  LIN {X -4860.893,Y -2029.899,Z -82.531,A 90.03341,B 0.00000,C 180.00000} ; retreat
  ; Step 3350, bar 1635
  LIN {X -4985.893,Y -2029.899,Z 855.478,A 90.03341,B 0.00000,C 180.00000} ; outside
  LIN {X -4985.893,Y -2029.899,Z -132.531,A 90.03341,B 0.00000,C 180.00000} ; preinsert
  LIN {X -4985.893,Y -2029.899,Z -382.531,A 90.03341,B 0.00000,C 180.00000} ; insert
  LIN {X -4985.893,Y -2029.899,Z -382.531,A 90.03341,B 0.00000,C 180.00000} ; release
  LIN {X -4985.893,Y -2029.899,Z -82.531,A 90.03341,B 0.00000,C 180.00000} ; retreat
  ; Step 3351, bar 1637
  LIN {X -5110.893,Y -2029.899,Z 855.478,A 90.03341,B 0.00000,C 180.00000} ; outside
  LIN {X -5110.893,Y -2029.899,Z -132.531,A 90.03341,B 0.00000,C 180.00000} ; preinsert
  LIN {X -5110.893,Y -2029.899,Z -382.531,A 90.03341,B 0.00000,C 180.00000} ; insert
  LIN {X -5110.893,Y -2029.899,Z -382.531,A 90.03341,B 0.00000,C 180.00000} ; release
  LIN {X -5110.893,Y -2029.899,Z -82.531,A 90.03341,B 0.00000,C 180.00000} ; retreat
  ; Step 3352, bar 1639
  LIN {X -5235.893,Y -2029.899,Z 855.478,A 90.03341,B 0.00000,C 180.00000} ; outside
  LIN {X -5235.893,Y -2029.899,Z -132.531,A 90.03341,B 0.00000,C 180.00000} ; preinsert
  LIN {X -5235.893,Y -2029.899,Z -382.531,A 90.03341,B 0.00000,C 180.00000} ; insert
  LIN {X -5235.893,Y -2029.899,Z -382.531,A 90.03341,B 0.00000,C 180.00000} ; release
  LIN {X -5235.893,Y -2029.899,Z -82.531,A 90.03341,B 0.00000,C 180.00000} ; retreat
  ; Step 3353, bar 1641
  LIN {X -5360.893,Y -2029.899,Z 855.478,A 90.03341,B 0.00000,C 180.00000} ; outside
  LIN {X -5360.893,Y -2029.899,Z -132.531,A 90.03341,B 0.00000,C 180.00000} ; preinsert
  LIN {X -5360.893,Y -2029.899,Z -382.531,A 90.03341,B 0.00000,C 180.00000} ; insert
  LIN {X -5360.893,Y -2029.899,Z -382.531,A 90.03341,B 0.00000,C 180.00000} ; release
  LIN {X -5360.893,Y -2029.899,Z -82.531,A 90.03341,B 0.00000,C 180.00000} ; retreat
  ; Step 3354, bar 1643
  LIN {X -5485.893,Y -2029.899,Z 855.478,A 90.03341,B 0.00000,C 180.00000} ; outside
  LIN {X -5485.893,Y -2029.899,Z -132.531,A 90.03341,B 0.00000,C 180.00000} ; preinsert
  LIN {X -5485.893,Y -2029.899,Z -382.531,A 90.03341,B 0.00000,C 180.00000} ; insert
  LIN {X -5485.893,Y -2029.899,Z -382.531,A 90.03341,B 0.00000,C 180.00000} ; release
  LIN {X -5485.893,Y -2029.899,Z -82.531,A 90.03341,B 0.00000,C 180.00000} ; retreat
  ; Step 3355, bar 1645
  LIN {X -5610.893,Y -2029.899,Z 855.478,A 90.03341,B 0.00000,C 180.00000} ; outside
  LIN {X -5610.893,Y -2029.899,Z -132.531,A 90.03341,B 0.00000,C 180.00000} ; preinsert
  LIN {X -5610.893,Y -2029.899,Z -382.531,A 90.03341,B 0.00000,C 180.00000} ; insert
  LIN {X -5610.893,Y -2029.899,Z -382.531,A 90.03341,B 0.00000,C 180.00000} ; release
  LIN {X -5610.893,Y -2029.899,Z -82.531,A 90.03341,B 0.00000,C 180.00000} ; retreat
  ; Step 3356, bar 1647
  LIN {X -5735.893,Y -2029.899,Z 855.478,A 90.03341,B 0.00000,C 180.00000} ; outside
  LIN {X -5735.893,Y -2029.899,Z -132.531,A 90.03341,B 0.00000,C 180.00000} ; preinsert
  LIN {X -5735.893,Y -2029.899,Z -382.531,A 90.03341,B 0.00000,C 180.00000} ; insert
  LIN {X -5735.893,Y -2029.899,Z -382.531,A 90.03341,B 0.00000,C 180.00000} ; release
  LIN {X -5735.893,Y -2029.899,Z -82.531,A 90.03341,B 0.00000,C 180.00000} ; retreat
  ; Step 3357, bar 1649
  LIN {X -5860.893,Y -2029.899,Z 855.478,A 90.03341,B 0.00000,C 180.00000} ; outside
  LIN {X -5860.893,Y -2029.899,Z -132.531,A 90.03341,B 0.00000,C 180.00000} ; preinsert
  LIN {X -5860.893,Y -2029.899,Z -382.531,A 90.03341,B 0.00000,C 180.00000} ; insert
  LIN {X -5860.893,Y -2029.899,Z -382.531,A 90.03341,B 0.00000,C 180.00000} ; release
  LIN {X -5860.893,Y -2029.899,Z -82.531,A 90.03341,B 0.00000,C 180.00000} ; retreat
  ; Step 3358, bar 1651
  LIN {X -6110.893,Y -2029.899,Z 855.478,A 90.03341,B 0.00000,C 180.00000} ; outside
  LIN {X -6110.893,Y -2029.899,Z -132.531,A 90.03341,B 0.00000,C 180.00000} ; preinsert
  LIN {X -6110.893,Y -2029.899,Z -382.531,A 90.03341,B 0.00000,C 180.00000} ; insert
  LIN {X -6110.893,Y -2029.899,Z -382.531,A 90.03341,B 0.00000,C 180.00000} ; release
  LIN {X -6110.893,Y -2029.899,Z -82.531,A 90.03341,B 0.00000,C 180.00000} ; retreat
  ; Step 3359, bar 1653
  LIN {X -6235.893,Y -2029.899,Z 855.478,A 90.03341,B 0.00000,C 180.00000} ; outside
  LIN {X -6235.893,Y -2029.899,Z -132.531,A 90.03341,B 0.00000,C 180.00000} ; preinsert
  LIN {X -6235.893,Y -2029.899,Z -382.531,A 90.03341,B 0.00000,C 180.00000} ; insert
  LIN {X -6235.893,Y -2029.899,Z -382.531,A 90.03341,B 0.00000,C 180.00000} ; release
  LIN {X -6235.893,Y -2029.899,Z -82.531,A 90.03341,B 0.00000,C 180.00000} ; retreat
  ; Step 3360, bar 1655
  LIN {X -6360.893,Y -2029.899,Z 855.478,A 90.03341,B 0.00000,C 180.00000} ; outside
  LIN {X -6360.893,Y -2029.899,Z -132.531,A 90.03341,B 0.00000,C 180.00000} ; preinsert
  LIN {X -6360.893,Y -2029.899,Z -382.531,A 90.03341,B 0.00000,C 180.00000} ; insert
  LIN {X -6360.893,Y -2029.899,Z -382.531,A 90.03341,B 0.00000,C 180.00000} ; release
  LIN {X -6360.893,Y -2029.899,Z -82.531,A 90.03341,B 0.00000,C 180.00000} ; retreat
  ; Step 3361, bar 1657
  LIN {X -6485.893,Y -2029.899,Z 855.478,A 90.03341,B 0.00000,C 180.00000} ; outside
  LIN {X -6485.893,Y -2029.899,Z -132.531,A 90.03341,B 0.00000,C 180.00000} ; preinsert
  LIN {X -6485.893,Y -2029.899,Z -382.531,A 90.03341,B 0.00000,C 180.00000} ; insert
  LIN {X -6485.893,Y -2029.899,Z -382.531,A 90.03341,B 0.00000,C 180.00000} ; release
  LIN {X -6485.893,Y -2029.899,Z -82.531,A 90.03341,B 0.00000,C 180.00000} ; retreat
  ; Step 3362, bar 1659
  LIN {X -6610.893,Y -2029.899,Z 855.478,A 90.03341,B 0.00000,C 180.00000} ; outside
  LIN {X -6610.893,Y -2029.899,Z -132.531,A 90.03341,B 0.00000,C 180.00000} ; preinsert
  LIN {X -6610.893,Y -2029.899,Z -382.531,A 90.03341,B 0.00000,C 180.00000} ; insert
  LIN {X -6610.893,Y -2029.899,Z -382.531,A 90.03341,B 0.00000,C 180.00000} ; release
  LIN {X -6610.893,Y -2029.899,Z -82.531,A 90.03341,B 0.00000,C 180.00000} ; retreat
  ; Step 3363, bar 1661
  LIN {X -6735.893,Y -2029.899,Z 855.478,A 90.03341,B 0.00000,C 180.00000} ; outside
  LIN {X -6735.893,Y -2029.899,Z -132.531,A 90.03341,B 0.00000,C 180.00000} ; preinsert
  LIN {X -6735.893,Y -2029.899,Z -382.531,A 90.03341,B 0.00000,C 180.00000} ; insert
  LIN {X -6735.893,Y -2029.899,Z -382.531,A 90.03341,B 0.00000,C 180.00000} ; release
  LIN {X -6735.893,Y -2029.899,Z -82.531,A 90.03341,B 0.00000,C 180.00000} ; retreat
  ; Step 3364, bar 1663
  LIN {X -6860.893,Y -2029.899,Z 855.478,A 90.03341,B 0.00000,C 180.00000} ; outside
  LIN {X -6860.893,Y -2029.899,Z -132.531,A 90.03341,B 0.00000,C 180.00000} ; preinsert
  LIN {X -6860.893,Y -2029.899,Z -382.531,A 90.03341,B 0.00000,C 180.00000} ; insert
  LIN {X -6860.893,Y -2029.899,Z -382.531,A 90.03341,B 0.00000,C 180.00000} ; release
  LIN {X -6860.893,Y -2029.899,Z -82.531,A 90.03341,B 0.00000,C 180.00000} ; retreat
  ; Step 3365, bar 1665
  LIN {X -6985.893,Y -2029.899,Z 855.478,A 90.03341,B 0.00000,C 180.00000} ; outside
  LIN {X -6985.893,Y -2029.899,Z -132.531,A 90.03341,B 0.00000,C 180.00000} ; preinsert
  LIN {X -6985.893,Y -2029.899,Z -382.531,A 90.03341,B 0.00000,C 180.00000} ; insert
  LIN {X -6985.893,Y -2029.899,Z -382.531,A 90.03341,B 0.00000,C 180.00000} ; release
  LIN {X -6985.893,Y -2029.899,Z -82.531,A 90.03341,B 0.00000,C 180.00000} ; retreat
  ; Step 3366, bar 1667
  LIN {X -7110.893,Y -2029.899,Z 855.478,A 90.03341,B 0.00000,C 180.00000} ; outside
  LIN {X -7110.893,Y -2029.899,Z -132.531,A 90.03341,B 0.00000,C 180.00000} ; preinsert
  LIN {X -7110.893,Y -2029.899,Z -382.531,A 90.03341,B 0.00000,C 180.00000} ; insert
  LIN {X -7110.893,Y -2029.899,Z -382.531,A 90.03341,B 0.00000,C 180.00000} ; release
  LIN {X -7110.893,Y -2029.899,Z -82.531,A 90.03341,B 0.00000,C 180.00000} ; retreat
  ; Step 3367, bar 1669
  LIN {X -7235.893,Y -2029.899,Z 855.478,A 90.03341,B 0.00000,C 180.00000} ; outside
  LIN {X -7235.893,Y -2029.899,Z -132.531,A 90.03341,B 0.00000,C 180.00000} ; preinsert
  LIN {X -7235.893,Y -2029.899,Z -382.531,A 90.03341,B 0.00000,C 180.00000} ; insert
  LIN {X -7235.893,Y -2029.899,Z -382.531,A 90.03341,B 0.00000,C 180.00000} ; release
  LIN {X -7235.893,Y -2029.899,Z -82.531,A 90.03341,B 0.00000,C 180.00000} ; retreat
  ; Step 3368, bar 1671
  LIN {X -7360.893,Y -2029.899,Z 855.478,A 90.03341,B 0.00000,C 180.00000} ; outside
  LIN {X -7360.893,Y -2029.899,Z -132.531,A 90.03341,B 0.00000,C 180.00000} ; preinsert
  LIN {X -7360.893,Y -2029.899,Z -382.531,A 90.03341,B 0.00000,C 180.00000} ; insert
  LIN {X -7360.893,Y -2029.899,Z -382.531,A 90.03341,B 0.00000,C 180.00000} ; release
  LIN {X -7360.893,Y -2029.899,Z -82.531,A 90.03341,B 0.00000,C 180.00000} ; retreat
  ; Step 3369, bar 1673
  LIN {X -7485.893,Y -2029.899,Z 855.478,A 90.03341,B 0.00000,C 180.00000} ; outside
  LIN {X -7485.893,Y -2029.899,Z -132.531,A 90.03341,B 0.00000,C 180.00000} ; preinsert
  LIN {X -7485.893,Y -2029.899,Z -382.531,A 90.03341,B 0.00000,C 180.00000} ; insert
  LIN {X -7485.893,Y -2029.899,Z -382.531,A 90.03341,B 0.00000,C 180.00000} ; release
  LIN {X -7485.893,Y -2029.899,Z -82.531,A 90.03341,B 0.00000,C 180.00000} ; retreat
  ; Step 3370, bar 1675
  LIN {X -7610.893,Y -2029.899,Z 855.478,A 90.03341,B 0.00000,C 180.00000} ; outside
  LIN {X -7610.893,Y -2029.899,Z -132.531,A 90.03341,B 0.00000,C 180.00000} ; preinsert
  LIN {X -7610.893,Y -2029.899,Z -382.531,A 90.03341,B 0.00000,C 180.00000} ; insert
  LIN {X -7610.893,Y -2029.899,Z -382.531,A 90.03341,B 0.00000,C 180.00000} ; release
  LIN {X -7610.893,Y -2029.899,Z -82.531,A 90.03341,B 0.00000,C 180.00000} ; retreat
  ; Step 3371, bar 1677
  LIN {X -7735.893,Y -2029.899,Z 855.478,A 90.03341,B 0.00000,C 180.00000} ; outside
  LIN {X -7735.893,Y -2029.899,Z -132.531,A 90.03341,B 0.00000,C 180.00000} ; preinsert
  LIN {X -7735.893,Y -2029.899,Z -382.531,A 90.03341,B 0.00000,C 180.00000} ; insert
  LIN {X -7735.893,Y -2029.899,Z -382.531,A 90.03341,B 0.00000,C 180.00000} ; release
  LIN {X -7735.893,Y -2029.899,Z -82.531,A 90.03341,B 0.00000,C 180.00000} ; retreat
  ; Step 3372, bar 1679
  LIN {X -7860.893,Y -2029.899,Z 855.478,A 90.03341,B 0.00000,C 180.00000} ; outside
  LIN {X -7860.893,Y -2029.899,Z -132.531,A 90.03341,B 0.00000,C 180.00000} ; preinsert
  LIN {X -7860.893,Y -2029.899,Z -382.531,A 90.03341,B 0.00000,C 180.00000} ; insert
  LIN {X -7860.893,Y -2029.899,Z -382.531,A 90.03341,B 0.00000,C 180.00000} ; release
  LIN {X -7860.893,Y -2029.899,Z -82.531,A 90.03341,B 0.00000,C 180.00000} ; retreat
  ; Step 3373, bar 1681
  LIN {X -7985.893,Y -2029.899,Z 855.478,A 90.03341,B 0.00000,C 180.00000} ; outside
  LIN {X -7985.893,Y -2029.899,Z -132.531,A 90.03341,B 0.00000,C 180.00000} ; preinsert
  LIN {X -7985.893,Y -2029.899,Z -382.531,A 90.03341,B 0.00000,C 180.00000} ; insert
  LIN {X -7985.893,Y -2029.899,Z -382.531,A 90.03341,B 0.00000,C 180.00000} ; release
  LIN {X -7985.893,Y -2029.899,Z -82.531,A 90.03341,B 0.00000,C 180.00000} ; retreat
  ; Step 3374, bar 1683
  LIN {X -8110.893,Y -2029.899,Z 855.478,A 90.03341,B 0.00000,C 180.00000} ; outside
  LIN {X -8110.893,Y -2029.899,Z -132.531,A 90.03341,B 0.00000,C 180.00000} ; preinsert
  LIN {X -8110.893,Y -2029.899,Z -382.531,A 90.03341,B 0.00000,C 180.00000} ; insert
  LIN {X -8110.893,Y -2029.899,Z -382.531,A 90.03341,B 0.00000,C 180.00000} ; release
  LIN {X -8110.893,Y -2029.899,Z -82.531,A 90.03341,B 0.00000,C 180.00000} ; retreat
  ; Step 3375, bar 1685
  LIN {X -8235.893,Y -2029.899,Z 855.478,A 90.03341,B 0.00000,C 180.00000} ; outside
  LIN {X -8235.893,Y -2029.899,Z -132.531,A 90.03341,B 0.00000,C 180.00000} ; preinsert
  LIN {X -8235.893,Y -2029.899,Z -382.531,A 90.03341,B 0.00000,C 180.00000} ; insert
  LIN {X -8235.893,Y -2029.899,Z -382.531,A 90.03341,B 0.00000,C 180.00000} ; release
  LIN {X -8235.893,Y -2029.899,Z -82.531,A 90.03341,B 0.00000,C 180.00000} ; retreat
  ; Step 3376, bar 1687
  LIN {X -8360.893,Y -2029.899,Z 855.478,A 90.03341,B 0.00000,C 180.00000} ; outside
  LIN {X -8360.893,Y -2029.899,Z -132.531,A 90.03341,B 0.00000,C 180.00000} ; preinsert
  LIN {X -8360.893,Y -2029.899,Z -382.531,A 90.03341,B 0.00000,C 180.00000} ; insert
  LIN {X -8360.893,Y -2029.899,Z -382.531,A 90.03341,B 0.00000,C 180.00000} ; release
  LIN {X -8360.893,Y -2029.899,Z -82.531,A 90.03341,B 0.00000,C 180.00000} ; retreat
  ; Step 3377, bar 1689
  LIN {X -8485.893,Y -2029.899,Z 855.478,A 90.03341,B 0.00000,C 180.00000} ; outside
  LIN {X -8485.893,Y -2029.899,Z -132.531,A 90.03341,B 0.00000,C 180.00000} ; preinsert
  LIN {X -8485.893,Y -2029.899,Z -382.531,A 90.03341,B 0.00000,C 180.00000} ; insert
  LIN {X -8485.893,Y -2029.899,Z -382.531,A 90.03341,B 0.00000,C 180.00000} ; release
  LIN {X -8485.893,Y -2029.899,Z -82.531,A 90.03341,B 0.00000,C 180.00000} ; retreat
  ; Step 3378, bar 1691
  LIN {X -8610.893,Y -2029.899,Z 855.478,A 90.03341,B 0.00000,C 180.00000} ; outside
  LIN {X -8610.893,Y -2029.899,Z -132.531,A 90.03341,B 0.00000,C 180.00000} ; preinsert
  LIN {X -8610.893,Y -2029.899,Z -382.531,A 90.03341,B 0.00000,C 180.00000} ; insert
  LIN {X -8610.893,Y -2029.899,Z -382.531,A 90.03341,B 0.00000,C 180.00000} ; release
  LIN {X -8610.893,Y -2029.899,Z -82.531,A 90.03341,B 0.00000,C 180.00000} ; retreat
  ; Step 3379, bar 1693
  LIN {X -8735.893,Y -2029.899,Z 855.478,A 90.03341,B 0.00000,C 180.00000} ; outside
  LIN {X -8735.893,Y -2029.899,Z -132.531,A 90.03341,B 0.00000,C 180.00000} ; preinsert
  LIN {X -8735.893,Y -2029.899,Z -382.531,A 90.03341,B 0.00000,C 180.00000} ; insert
  LIN {X -8735.893,Y -2029.899,Z -382.531,A 90.03341,B 0.00000,C 180.00000} ; release
  LIN {X -8735.893,Y -2029.899,Z -82.531,A 90.03341,B 0.00000,C 180.00000} ; retreat
  ; Step 3380, bar 1695
  LIN {X -8860.893,Y -2029.899,Z 855.478,A 90.03341,B 0.00000,C 180.00000} ; outside
  LIN {X -8860.893,Y -2029.899,Z -132.531,A 90.03341,B 0.00000,C 180.00000} ; preinsert
  LIN {X -8860.893,Y -2029.899,Z -382.531,A 90.03341,B 0.00000,C 180.00000} ; insert
  LIN {X -8860.893,Y -2029.899,Z -382.531,A 90.03341,B 0.00000,C 180.00000} ; release
  LIN {X -8860.893,Y -2029.899,Z -82.531,A 90.03341,B 0.00000,C 180.00000} ; retreat
  ; Step 3381, bar 1697
  LIN {X -8985.893,Y -2029.899,Z 855.478,A 90.03341,B 0.00000,C 180.00000} ; outside
  LIN {X -8985.893,Y -2029.899,Z -132.531,A 90.03341,B 0.00000,C 180.00000} ; preinsert
  LIN {X -8985.893,Y -2029.899,Z -382.531,A 90.03341,B 0.00000,C 180.00000} ; insert
  LIN {X -8985.893,Y -2029.899,Z -382.531,A 90.03341,B 0.00000,C 180.00000} ; release
  LIN {X -8985.893,Y -2029.899,Z -82.531,A 90.03341,B 0.00000,C 180.00000} ; retreat
  ; Step 3382, bar 1699
  LIN {X -9110.893,Y -2029.899,Z 855.478,A 90.03341,B 0.00000,C 180.00000} ; outside
  LIN {X -9110.893,Y -2029.899,Z -132.531,A 90.03341,B 0.00000,C 180.00000} ; preinsert
  LIN {X -9110.893,Y -2029.899,Z -382.531,A 90.03341,B 0.00000,C 180.00000} ; insert
  LIN {X -9110.893,Y -2029.899,Z -382.531,A 90.03341,B 0.00000,C 180.00000} ; release
  LIN {X -9110.893,Y -2029.899,Z -82.531,A 90.03341,B 0.00000,C 180.00000} ; retreat
  ; Step 3383, bar 1701
  LIN {X -9235.893,Y -2029.899,Z 855.478,A 90.03341,B 0.00000,C 180.00000} ; outside
  LIN {X -9235.893,Y -2029.899,Z -132.531,A 90.03341,B 0.00000,C 180.00000} ; preinsert
  LIN {X -9235.893,Y -2029.899,Z -382.531,A 90.03341,B 0.00000,C 180.00000} ; insert
  LIN {X -9235.893,Y -2029.899,Z -382.531,A 90.03341,B 0.00000,C 180.00000} ; release
  LIN {X -9235.893,Y -2029.899,Z -82.531,A 90.03341,B 0.00000,C 180.00000} ; retreat
  ; Step 3384, bar 1703
  LIN {X -9360.893,Y -2029.899,Z 855.478,A 90.03341,B 0.00000,C 180.00000} ; outside
  LIN {X -9360.893,Y -2029.899,Z -132.531,A 90.03341,B 0.00000,C 180.00000} ; preinsert
  LIN {X -9360.893,Y -2029.899,Z -382.531,A 90.03341,B 0.00000,C 180.00000} ; insert
  LIN {X -9360.893,Y -2029.899,Z -382.531,A 90.03341,B 0.00000,C 180.00000} ; release
  LIN {X -9360.893,Y -2029.899,Z -82.531,A 90.03341,B 0.00000,C 180.00000} ; retreat
  ; Step 3385, bar 1705
  LIN {X -9485.893,Y -2029.899,Z 855.478,A 90.03341,B 0.00000,C 180.00000} ; outside
  LIN {X -9485.893,Y -2029.899,Z -132.531,A 90.03341,B 0.00000,C 180.00000} ; preinsert
  LIN {X -9485.893,Y -2029.899,Z -382.531,A 90.03341,B 0.00000,C 180.00000} ; insert
  LIN {X -9485.893,Y -2029.899,Z -382.531,A 90.03341,B 0.00000,C 180.00000} ; release
  LIN {X -9485.893,Y -2029.899,Z -82.531,A 90.03341,B 0.00000,C 180.00000} ; retreat
  ; Step 3386, bar 1707
  LIN {X -9610.893,Y -2029.899,Z 855.478,A 90.03341,B 0.00000,C 180.00000} ; outside
  LIN {X -9610.893,Y -2029.899,Z -132.531,A 90.03341,B 0.00000,C 180.00000} ; preinsert
  LIN {X -9610.893,Y -2029.899,Z -382.531,A 90.03341,B 0.00000,C 180.00000} ; insert
  LIN {X -9610.893,Y -2029.899,Z -382.531,A 90.03341,B 0.00000,C 180.00000} ; release
  LIN {X -9610.893,Y -2029.899,Z -82.531,A 90.03341,B 0.00000,C 180.00000} ; retreat
  ; Step 3387, bar 1709
  LIN {X -9735.893,Y -2029.899,Z 855.478,A 90.03341,B 0.00000,C 180.00000} ; outside
  LIN {X -9735.893,Y -2029.899,Z -132.531,A 90.03341,B 0.00000,C 180.00000} ; preinsert
  LIN {X -9735.893,Y -2029.899,Z -382.531,A 90.03341,B 0.00000,C 180.00000} ; insert
  LIN {X -9735.893,Y -2029.899,Z -382.531,A 90.03341,B 0.00000,C 180.00000} ; release
  LIN {X -9735.893,Y -2029.899,Z -82.531,A 90.03341,B 0.00000,C 180.00000} ; retreat
  ; Step 3388, bar 1711
  LIN {X -9860.893,Y -2029.899,Z 855.478,A 90.03341,B 0.00000,C 180.00000} ; outside
  LIN {X -9860.893,Y -2029.899,Z -132.531,A 90.03341,B 0.00000,C 180.00000} ; preinsert
  LIN {X -9860.893,Y -2029.899,Z -382.531,A 90.03341,B 0.00000,C 180.00000} ; insert
  LIN {X -9860.893,Y -2029.899,Z -382.531,A 90.03341,B 0.00000,C 180.00000} ; release
  LIN {X -9860.893,Y -2029.899,Z -82.531,A 90.03341,B 0.00000,C 180.00000} ; retreat
  ; Step 3389, bar 1713
  LIN {X -10110.893,Y -2029.899,Z 855.478,A 90.03341,B 0.00000,C 180.00000} ; outside
  LIN {X -10110.893,Y -2029.899,Z -132.531,A 90.03341,B 0.00000,C 180.00000} ; preinsert
  LIN {X -10110.893,Y -2029.899,Z -382.531,A 90.03341,B 0.00000,C 180.00000} ; insert
  LIN {X -10110.893,Y -2029.899,Z -382.531,A 90.03341,B 0.00000,C 180.00000} ; release
  LIN {X -10110.893,Y -2029.899,Z -82.531,A 90.03341,B 0.00000,C 180.00000} ; retreat
  ; Step 3390, bar 1715
  LIN {X -10235.893,Y -2029.899,Z 855.478,A 90.03341,B 0.00000,C 180.00000} ; outside
  LIN {X -10235.893,Y -2029.899,Z -132.531,A 90.03341,B 0.00000,C 180.00000} ; preinsert
  LIN {X -10235.893,Y -2029.899,Z -382.531,A 90.03341,B 0.00000,C 180.00000} ; insert
  LIN {X -10235.893,Y -2029.899,Z -382.531,A 90.03341,B 0.00000,C 180.00000} ; release
  LIN {X -10235.893,Y -2029.899,Z -82.531,A 90.03341,B 0.00000,C 180.00000} ; retreat
  ; Step 3391, bar 1717
  LIN {X -10360.893,Y -2029.899,Z 855.478,A 90.03341,B 0.00000,C 180.00000} ; outside
  LIN {X -10360.893,Y -2029.899,Z -132.531,A 90.03341,B 0.00000,C 180.00000} ; preinsert
  LIN {X -10360.893,Y -2029.899,Z -382.531,A 90.03341,B 0.00000,C 180.00000} ; insert
  LIN {X -10360.893,Y -2029.899,Z -382.531,A 90.03341,B 0.00000,C 180.00000} ; release
  LIN {X -10360.893,Y -2029.899,Z -82.531,A 90.03341,B 0.00000,C 180.00000} ; retreat
  ; Step 3392, bar 1719
  LIN {X -10485.893,Y -2029.899,Z 855.478,A 90.03341,B 0.00000,C 180.00000} ; outside
  LIN {X -10485.893,Y -2029.899,Z -132.531,A 90.03341,B 0.00000,C 180.00000} ; preinsert
  LIN {X -10485.893,Y -2029.899,Z -382.531,A 90.03341,B 0.00000,C 180.00000} ; insert
  LIN {X -10485.893,Y -2029.899,Z -382.531,A 90.03341,B 0.00000,C 180.00000} ; release
  LIN {X -10485.893,Y -2029.899,Z -82.531,A 90.03341,B 0.00000,C 180.00000} ; retreat
  ; Step 3393, bar 1721
  LIN {X -10610.893,Y -2029.899,Z 855.478,A 90.03341,B 0.00000,C 180.00000} ; outside
  LIN {X -10610.893,Y -2029.899,Z -132.531,A 90.03341,B 0.00000,C 180.00000} ; preinsert
  LIN {X -10610.893,Y -2029.899,Z -382.531,A 90.03341,B 0.00000,C 180.00000} ; insert
  LIN {X -10610.893,Y -2029.899,Z -382.531,A 90.03341,B 0.00000,C 180.00000} ; release
  LIN {X -10610.893,Y -2029.899,Z -82.531,A 90.03341,B 0.00000,C 180.00000} ; retreat
  ; Step 3394, bar 1723
  LIN {X -10735.893,Y -2029.899,Z 855.478,A 90.03341,B 0.00000,C 180.00000} ; outside
  LIN {X -10735.893,Y -2029.899,Z -132.531,A 90.03341,B 0.00000,C 180.00000} ; preinsert
  LIN {X -10735.893,Y -2029.899,Z -382.531,A 90.03341,B 0.00000,C 180.00000} ; insert
  LIN {X -10735.893,Y -2029.899,Z -382.531,A 90.03341,B 0.00000,C 180.00000} ; release
  LIN {X -10735.893,Y -2029.899,Z -82.531,A 90.03341,B 0.00000,C 180.00000} ; retreat
  ; Step 3395, bar 1725
  LIN {X -10860.893,Y -2029.899,Z 855.478,A 90.03341,B 0.00000,C 180.00000} ; outside
  LIN {X -10860.893,Y -2029.899,Z -132.531,A 90.03341,B 0.00000,C 180.00000} ; preinsert
  LIN {X -10860.893,Y -2029.899,Z -382.531,A 90.03341,B 0.00000,C 180.00000} ; insert
  LIN {X -10860.893,Y -2029.899,Z -382.531,A 90.03341,B 0.00000,C 180.00000} ; release
  LIN {X -10860.893,Y -2029.899,Z -82.531,A 90.03341,B 0.00000,C 180.00000} ; retreat
  ; Step 3396, bar 1727
  LIN {X -10985.893,Y -2029.899,Z 855.478,A 90.03341,B 0.00000,C 180.00000} ; outside
  LIN {X -10985.893,Y -2029.899,Z -132.531,A 90.03341,B 0.00000,C 180.00000} ; preinsert
  LIN {X -10985.893,Y -2029.899,Z -382.531,A 90.03341,B 0.00000,C 180.00000} ; insert
  LIN {X -10985.893,Y -2029.899,Z -382.531,A 90.03341,B 0.00000,C 180.00000} ; release
  LIN {X -10985.893,Y -2029.899,Z -82.531,A 90.03341,B 0.00000,C 180.00000} ; retreat
  ; Step 3397, bar 1729
  LIN {X -11110.893,Y -2029.899,Z 855.478,A 90.03341,B 0.00000,C 180.00000} ; outside
  LIN {X -11110.893,Y -2029.899,Z -132.531,A 90.03341,B 0.00000,C 180.00000} ; preinsert
  LIN {X -11110.893,Y -2029.899,Z -382.531,A 90.03341,B 0.00000,C 180.00000} ; insert
  LIN {X -11110.893,Y -2029.899,Z -382.531,A 90.03341,B 0.00000,C 180.00000} ; release
  LIN {X -11110.893,Y -2029.899,Z -82.531,A 90.03341,B 0.00000,C 180.00000} ; retreat
  ; Step 3398, bar 1731
  LIN {X -11235.893,Y -2029.899,Z 855.478,A 90.03341,B 0.00000,C 180.00000} ; outside
  LIN {X -11235.893,Y -2029.899,Z -132.531,A 90.03341,B 0.00000,C 180.00000} ; preinsert
  LIN {X -11235.893,Y -2029.899,Z -382.531,A 90.03341,B 0.00000,C 180.00000} ; insert
  LIN {X -11235.893,Y -2029.899,Z -382.531,A 90.03341,B 0.00000,C 180.00000} ; release
  LIN {X -11235.893,Y -2029.899,Z -82.531,A 90.03341,B 0.00000,C 180.00000} ; retreat
  ; Step 3399, bar 1733
  LIN {X -11360.893,Y -2029.899,Z 855.478,A 90.03341,B 0.00000,C 180.00000} ; outside
  LIN {X -11360.893,Y -2029.899,Z -132.531,A 90.03341,B 0.00000,C 180.00000} ; preinsert
  LIN {X -11360.893,Y -2029.899,Z -382.531,A 90.03341,B 0.00000,C 180.00000} ; insert
  LIN {X -11360.893,Y -2029.899,Z -382.531,A 90.03341,B 0.00000,C 180.00000} ; release
  LIN {X -11360.893,Y -2029.899,Z -82.531,A 90.03341,B 0.00000,C 180.00000} ; retreat
  ; Step 3400, bar 1735
  LIN {X -11485.893,Y -2029.899,Z 855.478,A 90.03341,B 0.00000,C 180.00000} ; outside
  LIN {X -11485.893,Y -2029.899,Z -132.531,A 90.03341,B 0.00000,C 180.00000} ; preinsert
  LIN {X -11485.893,Y -2029.899,Z -382.531,A 90.03341,B 0.00000,C 180.00000} ; insert
  LIN {X -11485.893,Y -2029.899,Z -382.531,A 90.03341,B 0.00000,C 180.00000} ; release
  LIN {X -11485.893,Y -2029.899,Z -82.531,A 90.03341,B 0.00000,C 180.00000} ; retreat
  ; Step 3401, bar 1737
  LIN {X -11610.893,Y -2029.899,Z 855.478,A 90.03341,B 0.00000,C 180.00000} ; outside
  LIN {X -11610.893,Y -2029.899,Z -132.531,A 90.03341,B 0.00000,C 180.00000} ; preinsert
  LIN {X -11610.893,Y -2029.899,Z -382.531,A 90.03341,B 0.00000,C 180.00000} ; insert
  LIN {X -11610.893,Y -2029.899,Z -382.531,A 90.03341,B 0.00000,C 180.00000} ; release
  LIN {X -11610.893,Y -2029.899,Z -82.531,A 90.03341,B 0.00000,C 180.00000} ; retreat
  ; Step 3402, bar 1739
  LIN {X -11735.893,Y -2029.899,Z 855.478,A 90.03341,B 0.00000,C 180.00000} ; outside
  LIN {X -11735.893,Y -2029.899,Z -132.531,A 90.03341,B 0.00000,C 180.00000} ; preinsert
  LIN {X -11735.893,Y -2029.899,Z -382.531,A 90.03341,B 0.00000,C 180.00000} ; insert
  LIN {X -11735.893,Y -2029.899,Z -382.531,A 90.03341,B 0.00000,C 180.00000} ; release
  LIN {X -11735.893,Y -2029.899,Z -82.531,A 90.03341,B 0.00000,C 180.00000} ; retreat
  ; Step 3403, bar 1741
  LIN {X -11860.893,Y -2029.899,Z 855.478,A 90.03341,B 0.00000,C 180.00000} ; outside
  LIN {X -11860.893,Y -2029.899,Z -132.531,A 90.03341,B 0.00000,C 180.00000} ; preinsert
  LIN {X -11860.893,Y -2029.899,Z -382.531,A 90.03341,B 0.00000,C 180.00000} ; insert
  LIN {X -11860.893,Y -2029.899,Z -382.531,A 90.03341,B 0.00000,C 180.00000} ; release
  LIN {X -11860.893,Y -2029.899,Z -82.531,A 90.03341,B 0.00000,C 180.00000} ; retreat
  ; Step 3404, bar 1743
  LIN {X -11985.893,Y -2029.899,Z 855.478,A 90.03341,B 0.00000,C 180.00000} ; outside
  LIN {X -11985.893,Y -2029.899,Z -132.531,A 90.03341,B 0.00000,C 180.00000} ; preinsert
  LIN {X -11985.893,Y -2029.899,Z -382.531,A 90.03341,B 0.00000,C 180.00000} ; insert
  LIN {X -11985.893,Y -2029.899,Z -382.531,A 90.03341,B 0.00000,C 180.00000} ; release
  LIN {X -11985.893,Y -2029.899,Z -82.531,A 90.03341,B 0.00000,C 180.00000} ; retreat
  ; Step 3405, bar 1745
  LIN {X -12110.893,Y -2029.899,Z 855.478,A 90.03341,B 0.00000,C 180.00000} ; outside
  LIN {X -12110.893,Y -2029.899,Z -132.531,A 90.03341,B 0.00000,C 180.00000} ; preinsert
  LIN {X -12110.893,Y -2029.899,Z -382.531,A 90.03341,B 0.00000,C 180.00000} ; insert
  LIN {X -12110.893,Y -2029.899,Z -382.531,A 90.03341,B 0.00000,C 180.00000} ; release
  LIN {X -12110.893,Y -2029.899,Z -82.531,A 90.03341,B 0.00000,C 180.00000} ; retreat
  ; Step 3406, bar 1747
  LIN {X -12235.893,Y -2029.899,Z 855.478,A 90.03341,B 0.00000,C 180.00000} ; outside
  LIN {X -12235.893,Y -2029.899,Z -132.531,A 90.03341,B 0.00000,C 180.00000} ; preinsert
  LIN {X -12235.893,Y -2029.899,Z -382.531,A 90.03341,B 0.00000,C 180.00000} ; insert
  LIN {X -12235.893,Y -2029.899,Z -382.531,A 90.03341,B 0.00000,C 180.00000} ; release
  LIN {X -12235.893,Y -2029.899,Z -82.531,A 90.03341,B 0.00000,C 180.00000} ; retreat
  ; Step 3407, bar 1749
  LIN {X -12335.893,Y -2029.899,Z 855.478,A 90.03341,B 0.00000,C 180.00000} ; outside
  LIN {X -12335.893,Y -2029.899,Z -132.531,A 90.03341,B 0.00000,C 180.00000} ; preinsert
  LIN {X -12335.893,Y -2029.899,Z -382.531,A 90.03341,B 0.00000,C 180.00000} ; insert
  LIN {X -12335.893,Y -2029.899,Z -382.531,A 90.03341,B 0.00000,C 180.00000} ; release
  LIN {X -12335.893,Y -2029.899,Z -82.531,A 90.03341,B 0.00000,C 180.00000} ; retreat
  ; Step 3408, bar 1751
  LIN {X -12435.893,Y -2029.899,Z 855.478,A 90.03341,B 0.00000,C 180.00000} ; outside
  LIN {X -12435.893,Y -2029.899,Z -132.531,A 90.03341,B 0.00000,C 180.00000} ; preinsert
  LIN {X -12435.893,Y -2029.899,Z -382.531,A 90.03341,B 0.00000,C 180.00000} ; insert
  LIN {X -12435.893,Y -2029.899,Z -382.531,A 90.03341,B 0.00000,C 180.00000} ; release
  LIN {X -12435.893,Y -2029.899,Z -82.531,A 90.03341,B 0.00000,C 180.00000} ; retreat
  ; Step 3409, bar 1753
  LIN {X -12535.893,Y -2029.899,Z 855.478,A 90.03341,B 0.00000,C 180.00000} ; outside
  LIN {X -12535.893,Y -2029.899,Z -132.531,A 90.03341,B 0.00000,C 180.00000} ; preinsert
  LIN {X -12535.893,Y -2029.899,Z -382.531,A 90.03341,B 0.00000,C 180.00000} ; insert
  LIN {X -12535.893,Y -2029.899,Z -382.531,A 90.03341,B 0.00000,C 180.00000} ; release
  LIN {X -12535.893,Y -2029.899,Z -82.531,A 90.03341,B 0.00000,C 180.00000} ; retreat
  ; Step 3410, bar 1755
  LIN {X -12635.893,Y -2029.899,Z 855.478,A 90.03341,B 0.00000,C 180.00000} ; outside
  LIN {X -12635.893,Y -2029.899,Z -132.531,A 90.03341,B 0.00000,C 180.00000} ; preinsert
  LIN {X -12635.893,Y -2029.899,Z -382.531,A 90.03341,B 0.00000,C 180.00000} ; insert
  LIN {X -12635.893,Y -2029.899,Z -382.531,A 90.03341,B 0.00000,C 180.00000} ; release
  LIN {X -12635.893,Y -2029.899,Z -82.531,A 90.03341,B 0.00000,C 180.00000} ; retreat
  ; Step 3411, bar 1757
  LIN {X -12735.893,Y -2029.899,Z 855.478,A 90.03341,B 0.00000,C 180.00000} ; outside
  LIN {X -12735.893,Y -2029.899,Z -132.531,A 90.03341,B 0.00000,C 180.00000} ; preinsert
  LIN {X -12735.893,Y -2029.899,Z -382.531,A 90.03341,B 0.00000,C 180.00000} ; insert
  LIN {X -12735.893,Y -2029.899,Z -382.531,A 90.03341,B 0.00000,C 180.00000} ; release
  LIN {X -12735.893,Y -2029.899,Z -82.531,A 90.03341,B 0.00000,C 180.00000} ; retreat
  ; Step 3412, bar 1759
  LIN {X -12835.893,Y -2029.899,Z 855.478,A 90.03341,B 0.00000,C 180.00000} ; outside
  LIN {X -12835.893,Y -2029.899,Z -132.531,A 90.03341,B 0.00000,C 180.00000} ; preinsert
  LIN {X -12835.893,Y -2029.899,Z -382.531,A 90.03341,B 0.00000,C 180.00000} ; insert
  LIN {X -12835.893,Y -2029.899,Z -382.531,A 90.03341,B 0.00000,C 180.00000} ; release
  LIN {X -12835.893,Y -2029.899,Z -82.531,A 90.03341,B 0.00000,C 180.00000} ; retreat
  ; Step 3413, bar 1761
  LIN {X -12935.893,Y -2029.899,Z 855.478,A 90.03341,B 0.00000,C 180.00000} ; outside
  LIN {X -12935.893,Y -2029.899,Z -132.531,A 90.03341,B 0.00000,C 180.00000} ; preinsert
  LIN {X -12935.893,Y -2029.899,Z -382.531,A 90.03341,B 0.00000,C 180.00000} ; insert
  LIN {X -12935.893,Y -2029.899,Z -382.531,A 90.03341,B 0.00000,C 180.00000} ; release
  LIN {X -12935.893,Y -2029.899,Z -82.531,A 90.03341,B 0.00000,C 180.00000} ; retreat
  ; Step 3414, bar 1763
  LIN {X -13035.893,Y -2029.899,Z 855.478,A 90.03341,B 0.00000,C 180.00000} ; outside
  LIN {X -13035.893,Y -2029.899,Z -132.531,A 90.03341,B 0.00000,C 180.00000} ; preinsert
  LIN {X -13035.893,Y -2029.899,Z -382.531,A 90.03341,B 0.00000,C 180.00000} ; insert
  LIN {X -13035.893,Y -2029.899,Z -382.531,A 90.03341,B 0.00000,C 180.00000} ; release
  LIN {X -13035.893,Y -2029.899,Z -82.531,A 90.03341,B 0.00000,C 180.00000} ; retreat
  ; Step 3415, bar 1765
  LIN {X -13135.893,Y -2029.899,Z 855.478,A 90.03341,B 0.00000,C 180.00000} ; outside
  LIN {X -13135.893,Y -2029.899,Z -132.531,A 90.03341,B 0.00000,C 180.00000} ; preinsert
  LIN {X -13135.893,Y -2029.899,Z -382.531,A 90.03341,B 0.00000,C 180.00000} ; insert
  LIN {X -13135.893,Y -2029.899,Z -382.531,A 90.03341,B 0.00000,C 180.00000} ; release
  LIN {X -13135.893,Y -2029.899,Z -82.531,A 90.03341,B 0.00000,C 180.00000} ; retreat
  ; Step 3416, bar 1767
  LIN {X -13235.893,Y -2029.899,Z 855.478,A 90.03341,B 0.00000,C 180.00000} ; outside
  LIN {X -13235.893,Y -2029.899,Z -132.531,A 90.03341,B 0.00000,C 180.00000} ; preinsert
  LIN {X -13235.893,Y -2029.899,Z -382.531,A 90.03341,B 0.00000,C 180.00000} ; insert
  LIN {X -13235.893,Y -2029.899,Z -382.531,A 90.03341,B 0.00000,C 180.00000} ; release
  LIN {X -13235.893,Y -2029.899,Z -82.531,A 90.03341,B 0.00000,C 180.00000} ; retreat
  ; Step 3417, bar 1769
  LIN {X -13335.893,Y -2029.899,Z 855.478,A 90.03341,B 0.00000,C 180.00000} ; outside
  LIN {X -13335.893,Y -2029.899,Z -132.531,A 90.03341,B 0.00000,C 180.00000} ; preinsert
  LIN {X -13335.893,Y -2029.899,Z -382.531,A 90.03341,B 0.00000,C 180.00000} ; insert
  LIN {X -13335.893,Y -2029.899,Z -382.531,A 90.03341,B 0.00000,C 180.00000} ; release
  LIN {X -13335.893,Y -2029.899,Z -82.531,A 90.03341,B 0.00000,C 180.00000} ; retreat
  ; Step 3418, bar 1773
  LIN {X -13535.893,Y -2029.899,Z 855.478,A 90.03341,B 0.00000,C 180.00000} ; outside
  LIN {X -13535.893,Y -2029.899,Z -132.531,A 90.03341,B 0.00000,C 180.00000} ; preinsert
  LIN {X -13535.893,Y -2029.899,Z -382.531,A 90.03341,B 0.00000,C 180.00000} ; insert
  LIN {X -13535.893,Y -2029.899,Z -382.531,A 90.03341,B 0.00000,C 180.00000} ; release
  LIN {X -13535.893,Y -2029.899,Z -82.531,A 90.03341,B 0.00000,C 180.00000} ; retreat
  ; Step 3419, bar 1771
  LIN {X -13435.893,Y -2029.899,Z 855.478,A 90.03341,B 0.00000,C 180.00000} ; outside
  LIN {X -13435.893,Y -2029.899,Z -132.531,A 90.03341,B 0.00000,C 180.00000} ; preinsert
  LIN {X -13435.893,Y -2029.899,Z -382.531,A 90.03341,B 0.00000,C 180.00000} ; insert
  LIN {X -13435.893,Y -2029.899,Z -382.531,A 90.03341,B 0.00000,C 180.00000} ; release
  LIN {X -13435.893,Y -2029.899,Z -82.531,A 90.03341,B 0.00000,C 180.00000} ; retreat
  ; Step 3420, bar 1775
  LIN {X -13635.893,Y -2029.899,Z 855.478,A 90.03341,B 0.00000,C 180.00000} ; outside
  LIN {X -13635.893,Y -2029.899,Z -132.531,A 90.03341,B 0.00000,C 180.00000} ; preinsert
  LIN {X -13635.893,Y -2029.899,Z -382.531,A 90.03341,B 0.00000,C 180.00000} ; insert
  LIN {X -13635.893,Y -2029.899,Z -382.531,A 90.03341,B 0.00000,C 180.00000} ; release
  LIN {X -13635.893,Y -2029.899,Z -82.531,A 90.03341,B 0.00000,C 180.00000} ; retreat
  ; Step 3421, bar 1777
  LIN {X -13735.893,Y -2029.899,Z 855.478,A 90.03341,B 0.00000,C 180.00000} ; outside
  LIN {X -13735.893,Y -2029.899,Z -132.531,A 90.03341,B 0.00000,C 180.00000} ; preinsert
  LIN {X -13735.893,Y -2029.899,Z -382.531,A 90.03341,B 0.00000,C 180.00000} ; insert
  LIN {X -13735.893,Y -2029.899,Z -382.531,A 90.03341,B 0.00000,C 180.00000} ; release
  LIN {X -13735.893,Y -2029.899,Z -82.531,A 90.03341,B 0.00000,C 180.00000} ; retreat
  ; Step 3422, bar 1779
  LIN {X -13835.893,Y -2029.899,Z 855.478,A 90.03341,B 0.00000,C 180.00000} ; outside
  LIN {X -13835.893,Y -2029.899,Z -132.531,A 90.03341,B 0.00000,C 180.00000} ; preinsert
  LIN {X -13835.893,Y -2029.899,Z -382.531,A 90.03341,B 0.00000,C 180.00000} ; insert
  LIN {X -13835.893,Y -2029.899,Z -382.531,A 90.03341,B 0.00000,C 180.00000} ; release
  LIN {X -13835.893,Y -2029.899,Z -82.531,A 90.03341,B 0.00000,C 180.00000} ; retreat
  ; Step 3423, bar 1781
  LIN {X -14135.893,Y -2029.899,Z 855.478,A 90.03341,B 0.00000,C 180.00000} ; outside
  LIN {X -14135.893,Y -2029.899,Z -132.531,A 90.03341,B 0.00000,C 180.00000} ; preinsert
  LIN {X -14135.893,Y -2029.899,Z -382.531,A 90.03341,B 0.00000,C 180.00000} ; insert
  LIN {X -14135.893,Y -2029.899,Z -382.531,A 90.03341,B 0.00000,C 180.00000} ; release
  LIN {X -14135.893,Y -2029.899,Z -82.531,A 90.03341,B 0.00000,C 180.00000} ; retreat
  ; Step 3424, bar 1783
  LIN {X -14235.893,Y -2029.899,Z 855.478,A 90.03341,B 0.00000,C 180.00000} ; outside
  LIN {X -14235.893,Y -2029.899,Z -132.531,A 90.03341,B 0.00000,C 180.00000} ; preinsert
  LIN {X -14235.893,Y -2029.899,Z -382.531,A 90.03341,B 0.00000,C 180.00000} ; insert
  LIN {X -14235.893,Y -2029.899,Z -382.531,A 90.03341,B 0.00000,C 180.00000} ; release
  LIN {X -14235.893,Y -2029.899,Z -82.531,A 90.03341,B 0.00000,C 180.00000} ; retreat
END
